// TwinCAT 3 PLC project FMDataTests
// ProgramVersion: 3.1.4024.0
// libraries:
//   Data, * (TomasRompotl)
//   Strings, * (TomasRompotl)
//   Tc2_System, * (Beckhoff Automation GmbH)
//   Tc3_Module, * (Beckhoff Automation GmbH)
//   TcUnit, * (www.tcunit.org)
//   Types, * (TomasRompotl)
// project tree:
//   Comparison/ CompareAnyTypeTest.TcPOU, ComparisonFunctionsTest.TcPOU
//   Manipulate/ ManipulateFunctionsTest.TcPOU (not stored)
//   / PlcTask.TcTTO, PRG_Test.TcPOU, TestTableRow.TcDUT (not stored)
//   QuickSort/ QuickSortFunctionsTest.TcPOU
//   Sort/ SortFunctionsTest.TcPOU
//   TableSerialization/ TableDeserializerTest.TcPOU (not stored), TableSerializerTest.TcPOU (not stored)
// (motion and I/O tree: see PLC project fmtypestests)
// real-time tasks:
//   TASK FMTypesTestsTask: cycle T#1ms, priority 20, ADS port 350
//   TASK FMStringsTestsTask: cycle T#1ms, priority 21, ADS port 351
//   TASK FMDataTestsTask: cycle T#1ms, priority 22, ADS port 352
//   TASK FMMathTestsTask: cycle T#1ms, priority 23, ADS port 353
//   TASK FMTimeTestsTask: cycle T#1ms, priority 24, ADS port 354

CONFIGURATION FMDataTests
    RESOURCE PLC ON TwinCAT3
        TASK PlcTask(INTERVAL := T#1ms, PRIORITY := 22);
        PROGRAM PRG_Test WITH PlcTask : PRG_Test;
    END_RESOURCE
END_CONFIGURATION

// ---- PRG_Test.TcPOU
PROGRAM PRG_Test
VAR
	comparisonFunctionsTest : ComparisonFunctionsTest;
	compareAnyTypeTest : CompareAnyTypeTest;
	
	manipulateFunctionsTest : ManipulateFunctionsTest;
	quickSortFunctionsTest : QuickSortFunctionsTest;
	SortFunctionsTest : SortFunctionsTest;

	tableSerializerTest : TableSerializerTest;
	tableDeserializerTest : TableDeserializerTest;
END_VAR

TcUnit.RUN();

END_PROGRAM

// ---- Comparison/ComparisonFunctionsTest.TcPOU
FUNCTION_BLOCK ComparisonFunctionsTest EXTENDS TcUnit.FB_TestSuite
VAR
END_VAR

DataEqualsFunction();

METHOD DataEqualsFunction : BOOL
VAR
	data1 : INT;
	data2 : INT;
END_VAR
TcUnit.TEST('Data equals');

data1 := 42;
data2 := 0;

AssertEquals_BOOL(
	Expected := FALSE,
	Actual := DataEquals(data1, data2),
	Message := 'Data should not be equal');

data2 := data1;

AssertEquals_BOOL(
	Expected := TRUE,
	Actual := DataEquals(data1, data2),
	Message := 'Data should be equal');

TEST_FINISHED();
END_METHOD

END_FUNCTION_BLOCK

// ---- Comparison/CompareAnyTypeTest.TcPOU
FUNCTION_BLOCK CompareAnyTypeTest EXTENDS TcUnit.FB_TestSuite
VAR
END_VAR

IsEqualAnyTypeFunction();
IsGreaterThanAnyTypeFunction();
IsGreaterThanOrEqualAnyTypeFunction();
IsNotEqualAnyTypeFunction();
IsLessThanAnyTypeFunction();
IsLessThanOrEqualAnyTypeFunction();

METHOD IsEqualAnyTypeFunction : BOOL
VAR
	data1 : STRING;
	data2 : STRING;
END_VAR
TcUnit.TEST('Is equal any type');

ClearData(data1);
ClearData(data2);
data1 := '';
data2 := 'some test content';

AssertEquals_BOOL(
	Expected := FALSE,
	Actual := CompareAnyType(ToAnyType(data1), ComparisonOperator.Equal, ToAnyType(data2)),
	Message := 'Data should not be equal');

data1 := data2;

AssertEquals_BOOL(
	Expected := TRUE,
	Actual := CompareAnyType(ToAnyType(data1), ComparisonOperator.Equal, ToAnyType(data2)),
	Message := 'Data should be equal');

TEST_FINISHED();
END_METHOD

METHOD IsGreaterThanAnyTypeFunction : BOOL
VAR
	data1 : INT;
	data2 : INT;
END_VAR
TcUnit.TEST('Is greater then any type');

data1 := 5;
data2 := 5;

AssertEquals_BOOL(
	Expected := FALSE,
	Actual := CompareAnyType(ToAnyType(data1), ComparisonOperator.GreaterThan, ToAnyType(data2)),
	Message := 'data1 should not be greater then data2');

data1 := 10;

AssertEquals_BOOL(
	Expected := TRUE,
	Actual := CompareAnyType(ToAnyType(data1), ComparisonOperator.GreaterThan, ToAnyType(data2)),
	Message := 'data1 should be greater then data2');

TEST_FINISHED();
END_METHOD

METHOD IsGreaterThanOrEqualAnyTypeFunction : BOOL
VAR
	data1 : REAL;
	data2 : REAL;
END_VAR
TcUnit.TEST('Is greater then or equal any type');

data1 := 2.14;
data2 := 3.14;

AssertEquals_BOOL(
	Expected := FALSE,
	Actual := CompareAnyType(ToAnyType(data1), ComparisonOperator.GreaterThanOrEqual, ToAnyType(data2)),
	Message := 'data1 should not be greater or equal then data2');

data1 := 3.14;

AssertEquals_BOOL(
	Expected := TRUE,
	Actual := CompareAnyType(ToAnyType(data1), ComparisonOperator.GreaterThanOrEqual, ToAnyType(data2)),
	Message := 'data1 should be equal to data2');

data1 := 4.14;

AssertEquals_BOOL(
	Expected := TRUE,
	Actual := CompareAnyType(ToAnyType(data1), ComparisonOperator.GreaterThanOrEqual, ToAnyType(data2)),
	Message := 'data1 should be greater then data2');

TEST_FINISHED();
END_METHOD

METHOD IsLessThanAnyTypeFunction : BOOL
VAR
	data1 : INT;
	data2 : INT;
END_VAR
TcUnit.TEST('Is less then any type');

data1 := 5;
data2 := 5;

AssertEquals_BOOL(
	Expected := FALSE,
	Actual := CompareAnyType(ToAnyType(data1), ComparisonOperator.LessThan, ToAnyType(data2)),
	Message := 'data1 should not be less then data2');

data1 := 3;

AssertEquals_BOOL(
	Expected := TRUE,
	Actual := CompareAnyType(ToAnyType(data1), ComparisonOperator.LessThan, ToAnyType(data2)),
	Message := 'data1 should be less then data2');

TEST_FINISHED();
END_METHOD

METHOD IsLessThanOrEqualAnyTypeFunction : BOOL
VAR
	data1 : REAL;
	data2 : REAL;
END_VAR
TcUnit.TEST('Is less then or equal any type');

data1 := 4.14;
data2 := 3.14;

AssertEquals_BOOL(
	Expected := FALSE,
	Actual := CompareAnyType(ToAnyType(data1), ComparisonOperator.LessThanOrEqual, ToAnyType(data2)),
	Message := 'data1 should not be less or equal then data2');

data1 := 3.14;

AssertEquals_BOOL(
	Expected := TRUE,
	Actual := CompareAnyType(ToAnyType(data1), ComparisonOperator.LessThanOrEqual, ToAnyType(data2)),
	Message := 'data1 should be equal to data2');

data1 := 2.14;

AssertEquals_BOOL(
	Expected := TRUE,
	Actual := CompareAnyType(ToAnyType(data1), ComparisonOperator.LessThanOrEqual, ToAnyType(data2)),
	Message := 'data1 should be less then data2');

TEST_FINISHED();
END_METHOD

METHOD IsNotEqualAnyTypeFunction : BOOL
VAR
	data1 : STRING;
	data2 : STRING;
END_VAR
TcUnit.TEST('Is not equal any type');

ClearData(data1);
ClearData(data2);
data1 := 'some test content';
data2 := 'some test content';

AssertEquals_BOOL(
	Expected := FALSE,
	Actual := CompareAnyType(ToAnyType(data1), ComparisonOperator.NotEqual, ToAnyType(data2)),
	Message := 'Data should not be equal');

data1 := '';

AssertEquals_BOOL(
	Expected := TRUE,
	Actual := CompareAnyType(ToAnyType(data1), ComparisonOperator.NotEqual, ToAnyType(data2)),
	Message := 'Data should be equal');

TEST_FINISHED();
END_METHOD

END_FUNCTION_BLOCK

// ---- QuickSort/QuickSortFunctionsTest.TcPOU
FUNCTION_BLOCK QuickSortFunctionsTest EXTENDS TcUnit.FB_TestSuite
VAR
END_VAR

QuickSortREALFunction();

METHOD QuickSortREALFunction : BOOL
VAR
	data : ARRAY[0..4] OF REAL;
	expected : ARRAY[0..4] OF REAL;
END_VAR
TcUnit.TEST('QuickSort REAL');

data[0] := 3;
data[1] := 1;
data[2] := 2;
data[3] := 5;
data[4] := 4;

QuickSortREAL(data, 0, 4);

expected[0] := 1;
expected[1] := 2;
expected[2] := 3;
expected[3] := 4;
expected[4] := 5;

AssertArrayEquals_REAL(
	Expecteds := expected,
	Actuals := data,
	Delta := 0.1,
	Message := 'Array should be sorter');

TEST_FINISHED();
END_METHOD

END_FUNCTION_BLOCK

// ---- Sort/SortFunctionsTest.TcPOU
FUNCTION_BLOCK SortFunctionsTest EXTENDS TcUnit.FB_TestSuite
VAR
END_VAR

SortAnythingFunction();

METHOD SortAnythingFunction : BOOL
VAR
	data : ARRAY[0..4] OF TestTableRow;
	expected : ARRAY[0..4] OF TestTableRow;
	
	i : INT;
END_VAR
TcUnit.TEST('Sort anything');

ClearData(data);
ClearData(expected);

data[0].timestamp := T#3S;
data[0].value1 := 2;
data[0].value2 := 5.555;
data[0].description := 'some text';
data[1].timestamp := T#1S;
data[1].value1 := 8;
data[1].value2 := 3.14;
data[1].description := 'hello world';
data[2].timestamp := T#5S;
data[2].value1 := 15;
data[2].value2 := 9.876;
data[2].description := 'test data';
data[3].timestamp := T#2S;
data[3].value1 := 4;
data[3].value2 := 1.234;
data[3].description := 'sample entry';
data[4].timestamp := T#7S;
data[4].value1 := 11;
data[4].value2 := 6.789;
data[4].description := 'final record';

SortAnything(
	arr := data,
	firstElement := data[0],
	sortBy := data[0].value1,
	order := SortOrder.Descending
);

expected[0].timestamp := T#5S;
expected[0].value1 := 15;
expected[0].value2 := 9.876;
expected[0].description := 'test data';
expected[1].timestamp := T#7S;
expected[1].value1 := 11;
expected[1].value2 := 6.789;
expected[1].description := 'final record';
expected[2].timestamp := T#1S;
expected[2].value1 := 8;
expected[2].value2 := 3.14;
expected[2].description := 'hello world';
expected[3].timestamp := T#2S;
expected[3].value1 := 4;
expected[3].value2 := 1.234;
expected[3].description := 'sample entry';
expected[4].timestamp := T#3S;
expected[4].value1 := 2;
expected[4].value2 := 5.555;
expected[4].description := 'some text';

AssertEquals_BOOL(
	Expected := TRUE,
	Actual := DataEquals(data, expected),
	Message := 'Array should be sorted descending by value1 column');

TEST_FINISHED();
END_METHOD

END_FUNCTION_BLOCK
